ABB RobotStudio station: 吸盘.rsstn

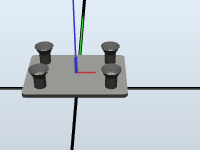
Station Station (saved by RobotStudio 6.8.8148.134)
Layout (positions relative to the parent item):
  - MyNewTool [mechanism] at (0, 0, 0) mm
      TCP MyNewTool at (0, 0, 50) mm
      links: 吸盘
  - 框架_1 [frame] at (0, 0, 50) mm
Attachment: 框架_1 is attached to MyNewTool / 吸盘
